Fanuc TP program (LS listing): UP112.LS

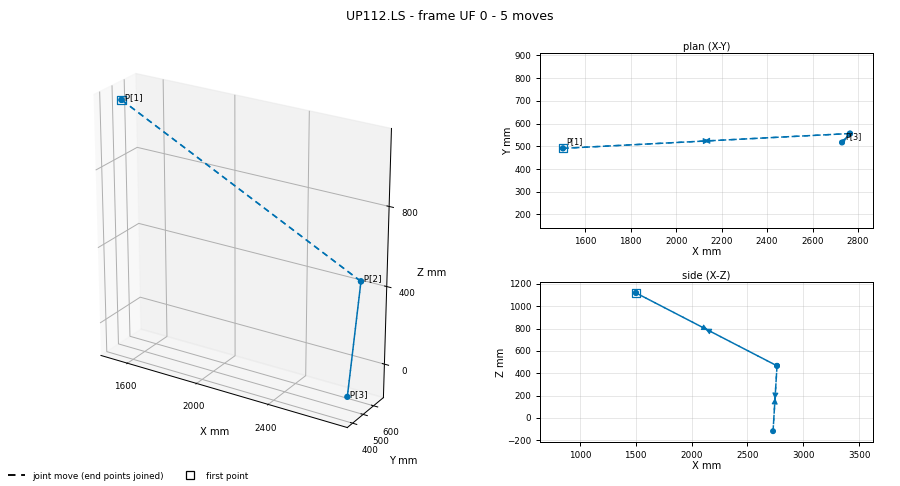
[picture p0: tool path of UP112.LS in frame UF 0, 5 of 5 moves have a stored position in this frame; points joined in program order, loops and branches not executed]
/PROG  UP112
/ATTR
OWNER		= AUROM;
COMMENT		= "Mant. G1";
PROG_SIZE	= 2740;
CREATE		= DATE 03-15-00  TIME 13:37:40;
MODIFIED	= DATE 17-02-24  TIME 04:54:42;
FILE_NAME	= ;
VERSION		= 0;
LINE_COUNT	= 9;
MEMORY_SIZE	= 4800;
PROTECT		= READ_WRITE;
TCD:  STACK_SIZE	= 500,
      TASK_PRIORITY	= 50,
      TIME_SLICE	= 0,
      BUSY_LAMP_OFF	= 0,
      ABORT_REQUEST	= 0,
      PAUSE_REQUEST	= 0;
DEFAULT_GROUP	= 1,1,1,1,*;
CONTROL_CODE	= 00000000 00000000;
/MN
   1:  UTOOL_NUM=1 ;
   2:  UFRAME_NUM=0 ;
   3:  PAYLOAD[1] ;
   4:J P[1] 100% CNT0 ACC100 TB    .10sec,P-SPS    ;
      1:  TC_ONLINE (ON) ;
      2:  DO[23]=OFF ;
      3:  CALL MAKRO050    ;
      4:  !Lib. de Herramientas ;
      5:  DO[80]=ON ;
      6:  DO[78]=OFF ;
      7:  DO[77]=ON ;
      8:  DO[75]=OFF ;
      9:  DO[74]=ON ;
     10:  DO[73]=ON ;
     11:  DO[71]=OFF ;
     12:  DO[70]=OFF ;
     13:  DO[69]=OFF ;
     14:  DO[68]=OFF ;
     15:  DO[67]=OFF ;
     16:  !Lib. de Anticolisiones ;
     17:  DO[41]=ON ;
     18:  DO[42]=ON ;
     19:  DO[43]=ON ;
     20:  DO[44]=ON ;
     21:  DO[45]=ON ;
     22:  DO[46]=ON ;
     23:  !Apagar Pos. Base ;
     24:  DO[15]=OFF ;
     25:  !Robot en Trayectoria ;
     26:  DO[16]=ON ;
     27:  WAIT (DI[23])    ;
     28:  DO[23]=ON ;
     29:  TC_ONLINE (M[2] AND M[30] AND M[31] AND M[35] AND M[37] AND M[39] AND M[41] AND M[43] AND M[95] AND M[96]) ;
       ------ ;
   5:J P[2] 100% CNT100 ACC100 TB   0.00sec,P-SPS    ;
      1:  TC_ONLINE (M[2] AND M[30] AND M[31] AND M[35] AND M[37] AND M[39] AND M[41] AND M[43] AND M[95] AND M[96]) ;
       ------ ;
   6:  !Pos. de Mantenimiento ;
   7:J P[3] 100% CNT0 ACC100 TB    .10sec,P-SPS    ;
      1:  TC_ONLINE (ON) ;
      2:  DO[23]=OFF ;
      3:  DO[17]=ON ;
      4:  GO[19]=1 ;
      5:  WAIT (DI[17])    ;
      6:  DO[17]=OFF ;
      7:  GO[19]=0 ;
      8:  WAIT (DI[23])    ;
      9:  DO[23]=ON ;
     10:  TC_ONLINE (M[2] AND M[30] AND M[31] AND M[35] AND M[37] AND M[39] AND M[41] AND M[43] AND M[95] AND M[96]) ;
       ------ ;
   8:J P[4] 100% CNT100 ACC100 TB   0.00sec,P-SPS    ;
      1:  TC_ONLINE (M[2] AND M[30] AND M[31] AND M[35] AND M[37] AND M[39] AND M[41] AND M[43] AND M[95] AND M[96]) ;
       ------ ;
   9:J P[5] 100% CNT0 ACC100 TB    .10sec,P-SPS    ;
      1:  TC_ONLINE (ON) ;
      2:  DO[23]=OFF ;
      3:  WAIT (DI[23])    ;
      4:  DO[23]=ON ;
      5:  TC_ONLINE (M[2] AND M[30] AND M[31] AND M[35] AND M[37] AND M[39] AND M[41] AND M[43] AND M[95] AND M[96]) ;
       ------ ;
/POS
P[1]{
   GP1:
	UF : 0, UT : 1,		CONFIG : 'N U T, 0, 0, 1',
	X =  1502.063  mm,	Y =   490.837  mm,	Z =  1119.244  mm,
	W =    -8.695 deg,	P =    50.167 deg,	R =     1.303 deg
   GP2:
	UF : 0, UT : 1,
	J1=   100.000  mm
   GP3:
	UF : 0, UT : 1,
	J1=     0.000  mm
   GP4:
	UF : 0, UT : 1,
	J1=     0.000  mm
};
P[2]{
   GP1:
	UF : 0, UT : 1,		CONFIG : 'F U T, 0, 0, 1',
	X =  2764.736  mm,	Y =   556.017  mm,	Z =   466.668  mm,
	W =    -3.827 deg,	P =    21.462 deg,	R =     5.565 deg
   GP2:
	UF : 0, UT : 1,
	J1=   100.000  mm
   GP3:
	UF : 0, UT : 1,
	J1=     0.000  mm
   GP4:
	UF : 0, UT : 1,
	J1=     0.000  mm
};
P[3]{
   GP1:
	UF : 0, UT : 1,		CONFIG : 'F U T, 0, 0, 0',
	X =  2729.144  mm,	Y =   516.354  mm,	Z =  -118.533  mm,
	W =     -.369 deg,	P =     1.338 deg,	R =     7.471 deg
   GP2:
	UF : 0, UT : 1,
	J1=   100.000  mm
   GP3:
	UF : 0, UT : 1,
	J1=     0.000  mm
   GP4:
	UF : 0, UT : 1,
	J1=     0.000  mm
};
P[4]{
   GP1:
	UF : 0, UT : 1,		CONFIG : 'F U T, 0, 0, 1',
	X =  2764.736  mm,	Y =   556.017  mm,	Z =   466.668  mm,
	W =    -3.827 deg,	P =    21.462 deg,	R =     5.565 deg
   GP2:
	UF : 0, UT : 1,
	J1=   100.000  mm
   GP3:
	UF : 0, UT : 1,
	J1=     0.000  mm
   GP4:
	UF : 0, UT : 1,
	J1=     0.000  mm
};
P[5]{
   GP1:
	UF : 0, UT : 1,		CONFIG : 'N U T, 0, 0, 1',
	X =  1502.063  mm,	Y =   490.837  mm,	Z =  1119.244  mm,
	W =    -8.695 deg,	P =    50.167 deg,	R =     1.303 deg
   GP2:
	UF : 0, UT : 1,
	J1=   100.000  mm
   GP3:
	UF : 0, UT : 1,
	J1=     0.000  mm
   GP4:
	UF : 0, UT : 1,
	J1=     0.000  mm
};
/END
